FUNCTION_BLOCK SLEEP
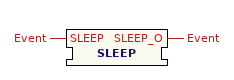
  EVENT_INPUT
    SLEEP;
  END_EVENT
  EVENT_OUTPUT
    SLEEP_O;
  END_EVENT
END_FUNCTION_BLOCK
